FUNCTION_BLOCK Feedback_FB
VAR_INPUT
	EN : BOOL;
	Command_1  : BOOL;
	Command_2  : BOOL;
	Command_3  : BOOL;
	Command_4  : BOOL;
	FeedbckDelyTime  : TIME;
END_VAR
VAR_OUTPUT
	ENO           : BOOL;
	Feedback_1    : BOOL;     
    Feedback_2    : BOOL;
	Feedback_3    : BOOL;     
    Feedback_4    : BOOL;
END_VAR
VAR
	fb1_Time       : TON;
	fb2_Time       : TON;
	fb3_Time       : TON;
	fb4_Time       : TON;
END_VAR

//FEEDBACK 1 DELAY

IF Command_1 THEN
	fb1_Time(IN := Command_1, PT :=FeedbckDelyTime);
	Feedback_1 := fb1_Time.Q;
	Feedback_2 := FALSE;
	Feedback_3 := FALSE;
	Feedback_4 := FALSE;
ELSE 
	fb1_Time(IN := FALSE);
END_IF;
	
//FEEDBACK 2 DELAY

IF Command_2 THEN
	fb2_Time(IN := Command_2, PT := FeedbckDelyTime);
	Feedback_2 := fb2_Time.Q;
	Feedback_1 := FALSE;
	Feedback_3 := FALSE;
	Feedback_4 := FALSE;
ELSE 
	fb2_Time(IN := FALSE);
END_IF;

//FEEDBACK 3 DELAY

IF Command_3 THEN
	fb3_Time(IN := Command_3, PT :=FeedbckDelyTime);
	Feedback_3 := fb3_Time.Q;
	Feedback_1 := FALSE;
	Feedback_2 := FALSE;
	Feedback_4 := FALSE;
ELSE 
	fb3_Time(IN := FALSE);
END_IF;
	
//FEEDBACK 4 DELAY

IF Command_4 THEN
	fb4_Time(IN := Command_4, PT := FeedbckDelyTime);
	Feedback_4 := fb4_Time.Q;
	Feedback_1 := FALSE;
	Feedback_2 := FALSE;
	Feedback_3 := FALSE;
ELSE 
	fb4_Time(IN := FALSE);
END_IF;

END_FUNCTION_BLOCK

(* stored: Version 1.1.0.1, ProductVersion 3.1.4024.16
   POU Feedback_FB: Id {fdea1f11-5f74-4592-899d-e2f99f283d0b}, SpecialFunc None *)
